SUBAPPLICATION AR_R_SUB (* Subtrahiert einen festen REAL-Subtrahenden von einem AR-Wert (OUT = IN - SUBTRAHEND; kein zweiter AR-Socket noetig - der Subtrahend wird per Parameter bei der Instanziierung eingebacken) *)
  (* Standard: 61499-2 *)
  (* Version 1.0, 2026-09-27, Franz Höpfinger, Meisterschulen am Ostbahnhof *)
  PACKAGE MyLib::sys;
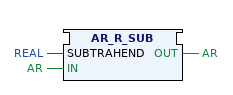
  VAR_INPUT
    SUBTRAHEND : REAL := REAL#0.0; (* Fester Subtrahend, ueber Parameter bei der Instanziierung gesetzt *)
  END_VAR
  SOCKETS
    IN : adapter::types::unidirectional::AR; (* Minuend-Wert *)
  END_SOCKETS
  PLUGS
    OUT : adapter::types::unidirectional::AR; (* IN - SUBTRAHEND *)
  END_PLUGS
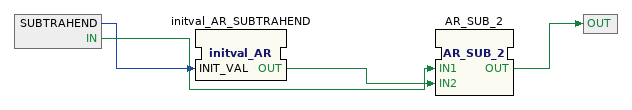
  FBS
    initval_AR_SUBTRAHEND : adapter::types::unidirectional::AR::initval::initval_AR;
    AR_SUB_2 : adapter::iec61131::arithmetic::AR_SUB_2;
  END_FBS
  DATA_CONNECTIONS
    SUBTRAHEND TO initval_AR_SUBTRAHEND.INIT_VAL;
  END_CONNECTIONS
  ADAPTER_CONNECTIONS
    IN TO AR_SUB_2.IN1;
    initval_AR_SUBTRAHEND.OUT TO AR_SUB_2.IN2;
    AR_SUB_2.OUT TO OUT;
  END_CONNECTIONS
END_SUBAPPLICATION
